(* Schneider Machine Expert - Basic project Test, file version 2.5.0.0 *)
(* CompanyInformations: WebSite=tyrone.zone *)
(* ProjectInformations: Name=Test, Description=Testing git for versioning control *)
(* UserInformations: FirstName=Tyrone, Country=New Zealand *)

HARDWARE
  Cpu 0: TM221CE24T
  EthernetConfiguration: NetworkName=M221, IpAllocationMode=FixedAddress, IpAddress=0.0.0.0, SubnetMask=0.0.0.0
  SerialLineConfiguration: Baud=Baud19200, Parity=ParityEven, DataBits=DataBits8, StopBits=StopBits1, PhysicalMedium=PhysicalMediumRs485, TransmissionMode=TransmissionModeModbusRtu, SlaveId=1, Addressing=SlaveAddressing
  MastTask: UsePeriodScanMode=false, PeriodScan=100
  FastTask: Period=255
  CpuBehavior: StartingMode=StartAsPreviousState, AutoSaveRamOnEeprom=true, WatchdogPeriod=250

SYMBOLS  (address, symbol, comment, settings)
  %I0.0       "Input"
  %Q0.0       "Output"

GRAFCET Grafcet POU
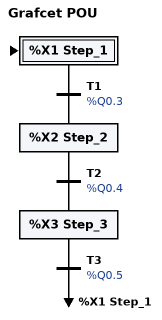
  INITIAL_STEP %X1  (* Step_1 *)
  STEP %X2  (* Step_2 *)
  STEP %X3  (* Step_3 *)
  TRANSITION T1 FROM %X1 TO %X2 := %Q0.3;
  TRANSITION T2 FROM %X2 TO %X3 := %Q0.4;
  TRANSITION T3 FROM %X3 TO %X1 := %Q0.5;

POU POU Name  (* POU Comment *)
  (* SectionNumber=1 *)

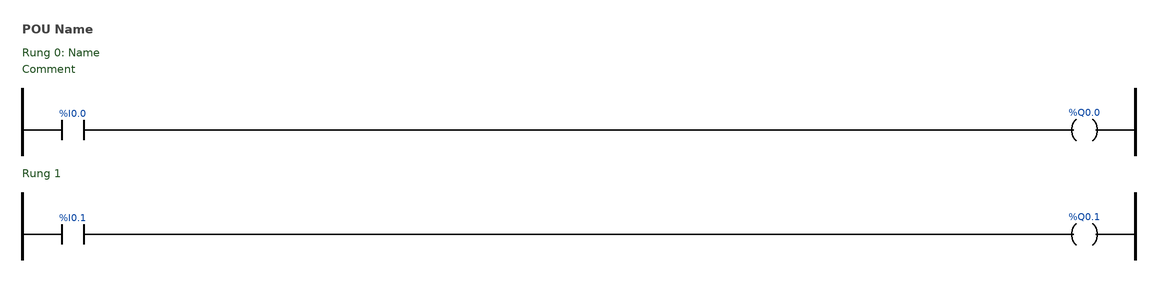

// Rung 0: Name
// Comment
  LD %I0.0
  ST %Q0.0
  // as ST:
  //   %Q0.0 := %I0.0;

// Rung 1
  LD %I0.1
  ST %Q0.1
  // as ST:
  //   %Q0.1 := %I0.1;

POU New POU
  (* SectionNumber=2 *)

// Rung 2
  LD %I0.2
  ST %Q0.2
  // as ST:
  //   %Q0.2 := %I0.2;

STEP %X1 Step_1
  (* SectionNumber=3, StepNumber=1 *)

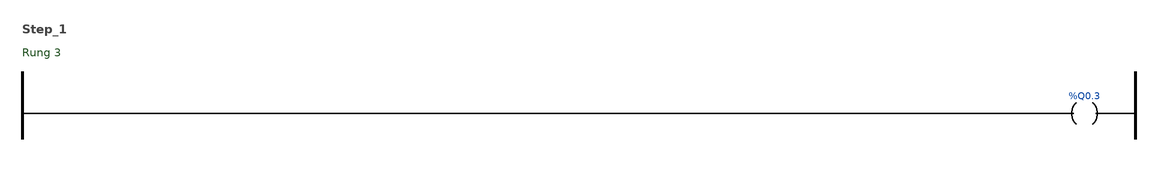

// Rung 3
  LD 1
  ST %Q0.3
  // as ST:
  //   %Q0.3 := TRUE;

STEP %X2 Step_2
  (* SectionNumber=4, StepNumber=2 *)

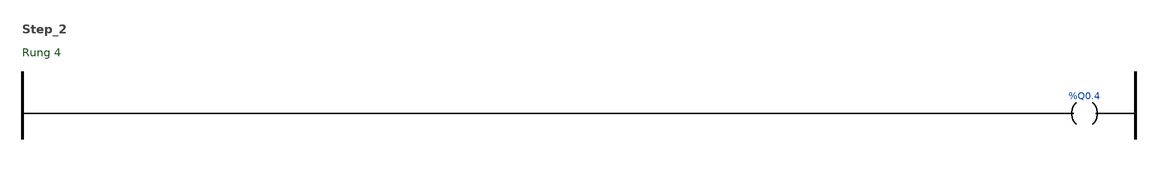

// Rung 4
  LD 1
  ST %Q0.4
  // as ST:
  //   %Q0.4 := TRUE;

STEP %X3 Step_3
  (* SectionNumber=5, StepNumber=3 *)

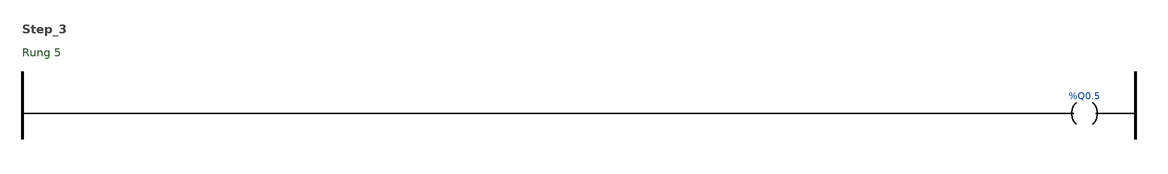

// Rung 5
  LD 1
  ST %Q0.5
  // as ST:
  //   %Q0.5 := TRUE;

TRANSITION T1 (%X1 -> %X2) 
  (* SectionNumber=0 *)

// Rung 6: Tr1
  LD %Q0.3
  ENDT
  // as ST:
  //   TRANSITION := %Q0.3;

TRANSITION T2 (%X2 -> %X3) 
  (* SectionNumber=0 *)

// Rung 7: Tr2
  LD %Q0.4
  ENDT
  // as ST:
  //   TRANSITION := %Q0.4;

TRANSITION T3 (%X3 -> %X1) 
  (* SectionNumber=0 *)

// Rung 8: Tr3
  LD %Q0.5
  ENDT
  // as ST:
  //   TRANSITION := %Q0.5;
